// TIA Portal V19 export
DATA_BLOCK "MFG PROCESS"   // DB24
{ S7_Optimized_Access := 'TRUE' }
// stored: MemoryReserve 100
   VAR
      MFG : Int;
   END_VAR
BEGIN
END_DATA_BLOCK
